// TIA Portal V18 export
DATA_BLOCK "FC51_Control_DB"   // DB1
// stored: InstanceOfName FC51_Control, InstanceOfType FB
"FC51_Control"
   // VAR_INPUT
   //    I_Start : Bool;
   //    I_Frequency : Real;
   //    I_Alarm_Confirm : Bool;
   // END_VAR
   // VAR
   //    FB_Always_True : Bool;
   //    Frequency_Trans_Instance { ExternalAccessible := 'False'; ExternalVisible := 'False'; ExternalWritable := 'False'} : "Frequency_Trans";
   //    FC51_Modbus_Com_Instance { S7_SetPoint := 'True'} : "FC51_Modbus_Com";
   // END_VAR
BEGIN
END_DATA_BLOCK
